// TIA Portal V19 export
FUNCTION "FC_FPosFree" : Void   // FC37, STL
TITLE = FPosFree weitergeben
{ S7_Optimized_Access := 'FALSE' }
AUTHOR : MS
// stored: AutoNumber false
   VAR_INPUT
      WT_Nr : Int;
      Pos : USInt;   // Position in der WT ist (sein sollte)
      am_FW_QT : Bool;
   END_VAR
   VAR_TEMP
      savAR1 : DWord;
      savAR2 : DWord;
      WT_DB : Word;
      ChkPos : Int;
      B_PNTR : Int;
      newB_PNTR : Int;
      Adresse : DWord;
      Ziel_1 : Int;
      Leng_1 : Int;
      Ziel_2 : Int;
      Leng_2 : Int;
      WT_Typ : Byte;
      Pos_Typ : Byte;
      Reihe : Byte;
      Typ_chk : Bool;   // 0=einfacher Check 10h 20h, 1=detailcheck 11h 12h usw.
      p_fnd : Bool;
      free : Bool;
      fPosfree : Bool;
   END_VAR
BEGIN

NETWORK
TITLE = Register retten
      A     "DB_ANLAGE".config.Anl_getaktet;
      BEC;

// --------------------------------
// Register retten
// --------------------------------
      TAR1;
      T     #savAR1;
      TAR2;
      T     #savAR2;

NETWORK
TITLE = Initialisierung
      L     #WT_Nr;
      +     100;
      T     #WT_DB;

      L     0;
      T     #Reihe;

NETWORK
TITLE = Zielposition prüfen
//-------------------------------------------
//Position prüfen
//-------------------------------------------
      L     #Pos;
      L     "DB_POS".LENG;
      *D;
      L     "DB_POS".Offset;
      +D;
      SLD   3;
      LAR1;
      OPN   "DB_POS";
//Pos mit anderem WT belegt --> Abbruch
      L     DBB [AR1, P#36.0];
      L     #WT_Nr;
      <>I;
      A(;
      L     DBB [AR1, P#36.0];
      L     0;
      <>I;
      );
      JC    raus;

//Pos gesperrt --> Abbruch
      L     DBB [AR1, P#0.0];  //PosTyp
      L     10;  //Typ QT
      <>I;
      A     DBX [AR1, P#9.1];  //notFG_in
      AN    #am_FW_QT;
      O     DBX [AR1, P#7.0];  //Sperre_in
      O     DBX [AR1, P#7.2];  //Sperre_out
      JC    raus;

      A     #am_FW_QT;
      S     DBX [AR1, P#6.3];  //reserviertes Ziel
      L     #WT_Nr;
      T     DBB [AR1, P#36.0];

      AN    DBX [AR1, P#9.3];  //"DB_POS".POS[0].fPosfree
      JC    raus;


NETWORK
TITLE = Initialisierung
//-------------------------------------------
//WT-Typ bestimmen (Trommel, Gestell usw.)
//-------------------------------------------
      A     "DB_ANLAGE".config.TypChckDetail;
      =     #Typ_chk;

      OPN   DB [#WT_DB];
      L     %DBB35;  //"DB_WT1".WT_Typ
      T     #WT_Typ;

//-------------------------------------------
//WT-DB öffnen
//-------------------------------------------
      L     #WT_Nr;
      L     100;
      +I;
      T     #WT_DB;
      OPN   DI [#WT_DB];
//-------------------------------------------
//Reihe bestimmen
//-------------------------------------------
      L     0;
      L     %DIB21;  //"DB_WT1".Ziel_Pos_WT
      <>I;
      JC    Reih;
      L     0;
      L     %DIB15;  //"DB_WT1".POS
      ==I;
      JC    nRh;
Reih: L     "DB_POS".LENG;
      *D;
      L     "DB_POS".Offset;
      +D;
      SLD   3;
      LAR1;
      OPN   "DB_POS";
      L     DBB [AR1, P#4.0];  //"DB_POS".POS[0].Reihe
      T     #Reihe;
//-------------------------------------------
//Befehlspointer laden
//-------------------------------------------
nRh:  L     %DIW48;  //"DB_WT1".B_PNTER
      T     #B_PNTR;

//-------------------------------------------
//Pointerkorrektur falls erforderlich
//z.Bsp: am FW oder bei DBB36<>0
//-------------------------------------------
      AN    #am_FW_QT;
      JC    endI;

      CALL  "FC_Pointer_Tech"
      ( Befehl       := #B_PNTR,
        Position     := #Pos,
        WT_Nr        := #WT_DB,
        p_fnd        := #p_fnd,
        new_Bef_Pntr := #newB_PNTR
      );

      AN    #p_fnd;
      JC    endI;

      L     #newB_PNTR;
      +     1;
      T     #B_PNTR;

endI: NOP   0;

NETWORK
TITLE = Zwngsziel prüfen
      L     #Pos;
      SLD   3;
      T     #Adresse;
      OPN   "DB_Zwangsziel";
      L     0;
      L     DBB [#Adresse];
      ==I;
      JC    endZ;
      T     #ChkPos;
      L     "DB_POS".LENG;
      *D;
      L     "DB_POS".Offset;
      +D;
      SLD   3;
      LAR1;
      OPN   "DB_POS";
      L     0;
      L     DBB [AR1, P#35.0];  //"DB_POS".POS[0].Reihe
      ==I;
      O(;
      L     #WT_Nr;
      ==I;
      );
      JC    endZ;
      L     0;
      L     DBB [AR1, P#36.0];  //"DB_POS".POS[0].Reihe
      <>I;
      A(;
      L     #WT_Nr;
      <>I;
      );
      JC    raus;

endZ: NOP   0;

NETWORK
TITLE = fPosfree-Schleife vor

      L     #B_PNTR;
retV: T     #newB_PNTR;
      OPN   DB [#WT_DB];
      L     %DBW0;  //"DB_WT1".ANZAHL
      >I;
      JC    raus;
      L     #newB_PNTR;
      L     %DBW4;  //"DB_WT1".LENG
      *D;
      L     %DBW2;  //"DB_WT1".OFFSET
      +D;
      SLD   3;
      LAR1;
      L     0;  //Ende Suchbereich
      L     DBB [AR1, P#0.0];  //"DB_WT1".Befehl[0].Kennung
      ==I;
      JC    raus;
//bis 220 normal
      L     DBB [AR1, P#0.0];  //Cmd
      L     220;
      <I;
      JC    chkB;
//220-229 (DC..E5) Variante
      L     DBB [AR1, P#0.0];  //Cmd
      L     230;
      <I;
      JC    VarB;
//230-235 (E6..EB) Quertransport
      L     DBB [AR1, P#0.0];  //Cmd
      L     240;
      <I;
      JC    nexV;
//240-249 (F0..F9) Gruppenfahrt
//250-252 (FA..FC) Speicherfahrt
      L     DBB [AR1, P#0.0];  //Cmd
      L     254;
      <I;
      JC    raus;
//254 (FE) Kontrolle//Sonderbefehle überspringen
//255 (FF) Trockner einschalten
      JU    nexV;

//Variantenbefehl
VarB: L     DBB [AR1, P#0.0];  //Cmd
      L     220;
      -I;
      T     #Ziel_1;
      +     1;
      L     "DB_Variantenbefehl".Anzahl_Varianten;
      >I;  //ungültige Variantengruppe
      JC    raus;

      OPN   DB [#WT_DB];
      L     DBW [AR1, P#6.0];  //Parameterpointer
      SLD   3;
      T     #Adresse;
      L     0;  //Variante überspringen
      L     DBB [#Adresse];  //Variante
      ==I;
      JC    nexV;
      T     #Ziel_2;
      L     "DB_Variantenbefehl".max_Var;
      >I;  //ungültige Variante
      JC    raus;

      L     #Ziel_1;
      L     "DB_Variantenbefehl".max_Var;
      *D;
      L     "DB_Variantenbefehl".Offset;
      +D;
      L     #Ziel_2;
      +D;
      +     -1;  //Korrektur Variante
      SLD   3;
      OPN   "DB_Variantenbefehl";
      T     #Adresse;

      L     DBB [#Adresse];  //Ziel_Position
VarC: T     #Ziel_1;
      L     1;
      T     #Leng_1;
      L     0;
      T     #Ziel_2;
      T     #Leng_2;

test: CALL  "FC_fPosfreePos"
      ( WT_Nr      := #WT_Nr,
        WT_Typ     := #WT_Typ,
        TypChk     := #Typ_chk,
        free       := #free,
        fPosfree   := #fPosfree,
        Zwangsziel := #ChkPos,
        Ziel_1     := #Ziel_1,
        leng_1     := #Leng_1,
        Ziel_2     := #Ziel_2,
        leng_2     := #Leng_2,
        Reihe      := #Reihe
      );

      AN    #free;
      JC    zrk;

      AN    #fPosfree;
      JC    raus;

      L     0;
      L     #ChkPos;
      ==I;
      JC    nexV;
      JU    VarC;

//Normaler Befehl
chkB: OPN   DB [#WT_DB];
      L     DBB [AR1, P#1.0];  //Ziel_1
      T     #Ziel_1;
      L     DBB [AR1, P#2.0];  //leng_1
      T     #Leng_1;
      L     DBB [AR1, P#3.0];  //Ziel_2
      T     #Ziel_2;
      L     DBB [AR1, P#4.0];  //leng_2
      T     #Leng_2;
      JU    test;

nexV: L     #newB_PNTR;
      +     1;
      JU    retV;


NETWORK
TITLE = Spuren löschen, wenn fPosfree-Strecke nicht frei
zrk:  NOP   0;
//evtl. alle Pos mit Dbb36 == WT_Nr löschen


NETWORK
TITLE = Adressregister wiederherstellen
//--------------------------------------
//Adressregister wiederherstellen
//--------------------------------------
raus: L     #savAR1;
      LAR1;
      L     #savAR2;
      LAR2;
END_FUNCTION
